// TIA Portal V20 export
DATA_BLOCK "DB_LoaderShuttle1"   // DB204
// stored: AutoNumber false, InstanceOfName FB_LoaderShuttle1, InstanceOfType FB
"FB_LoaderShuttle1"
   // VAR_INPUT
   //    iGripperReserved : Bool;
   //    iGripperReleased : Bool;
   //    iShuttleMoving : Bool;
   //    iShuttleInPos : Bool;
   //    iAxisV_Moving : Bool;
   //    iAxisV_InPos : Bool;
   //    iAxisW_Moving : Bool;
   //    iAxisW_InPos : Bool;
   // END_VAR
   // VAR_OUTPUT
   //    oExtGateOpenReq : Bool;
   //    oExtGateCloseReq : Bool;
   //    oIntGateOpenReq : Bool;
   //    oIntGateCloseReq : Bool;
   //    oLoadGripperCloseReq : Bool;
   //    oUnloadGripperOpenReq : Bool;
   //    oBlowingReq : Bool;
   //    oShuttleStartReq : Bool;
   //    oShuttlePosSetPoint : Real;
   //    oAxisVStartReq : Bool;
   //    oAxisVPosSetPoint : Real;
   //    oAxisWStartReq : Bool;
   //    oAxisWPosSetPoint : Real;
   // END_VAR
   // VAR
   //    sMain : "FB_Main";
   //    sShuttleInt { S7_SetPoint := 'True'} : "FB_ShuttleInt";
   //    sShuttleExt { S7_SetPoint := 'True'} : "FB_ShuttleExt";
   //    sControlIn { S7_SetPoint := 'True'} : "FB_PartControl";
   //    sControlOut { S7_SetPoint := 'True'} : "FB_PartControl";
   //    sBlowing { S7_SetPoint := 'True'} : "FB_Blowing";
   //    sIntLoadUnload { S7_SetPoint := 'True'} : "FB_IntLoadUnload";
   //    sExtLoadUnload { S7_SetPoint := 'True'} : "FB_ExtLoadUnload";
   //    sBwLoadUnload { S7_SetPoint := 'True'} : "FB_BwLoadUnload";
   //    sBwControlIn { S7_SetPoint := 'True'} : "FB_BwControl";
   //    sActPartControlIn { S7_SetPoint := 'True'} : "FB_ActControl";
   //    sActPartControlOut { S7_SetPoint := 'True'} : "FB_ActControl";
   //    sActBwControlIn { S7_SetPoint := 'True'} : "FB_ActControl";
   //    sIntLoadUnloadOP { S7_SetPoint := 'True'} : "FB_IntLoadUnloadOP";
   //    sBwConsecutiveCtrl { S7_SetPoint := 'True'} : "FB_Consecutive";
   //    sShuttlePosInt { S7_SetPoint := 'True'} : Bool;
   //    sShuttlePosSas : Bool;
   //    sShuttlePosExt : Bool;
   //    sGripper_OK : Bool;
   //    sExtLoaderInSafePos : Bool;
   //    sIntLoaderInSafePos : Bool;
   //    sBwLoaderInSafePos : Bool;
   //    sRT_PartControlInMissing : R_TRIG;
   //    sRT_PartControlInExtra : R_TRIG;
   //    sRT_PartControlOutMissing : R_TRIG;
   //    sRT_PartControlOutExtra : R_TRIG;
   //    sRT_BwControlInMissing : R_TRIG;
   //    sRT_BwControlInExtra : R_TRIG;
   //    sStepPauseSeq { S7_SetPoint := 'True'} : Bool;
   // END_VAR
BEGIN
END_DATA_BLOCK
